(* PLC project Unnamed, Unknown Unnamed 1 *)
(* stored: creationDateTime 2021-11-19T07:51:07, modificationDateTime 2021-11-26T10:24:18 *)

PROGRAM program0
  VAR
    Start : BOOL;
    Stop : BOOL;
    ConveyorBelt : BOOL;
    A : BOOL;
    B : BOOL;
    TON0 : TON;
    TON1 : TON;
    DetectCan : BOOL;
    DetectCap : BOOL;
    Wait1 : BOOL;
    TON2 : TON;
    Stop1 : BOOL;
    Detect : BOOL;
    ShootInkJet : BOOL;
    Wait2 : BOOL;
    TON3 : TON;
    Stop2 : BOOL;
    CountCan : BOOL;
    CTU0 : CTU;
    StartPalletizer : BOOL;
    CTU1 : CTU;
  END_VAR
  VAR  (* added by the conversion: wires and edge detectors of the diagram *)
    R_TRIG1 : R_TRIG;
    R_TRIG2 : R_TRIG;
  END_VAR

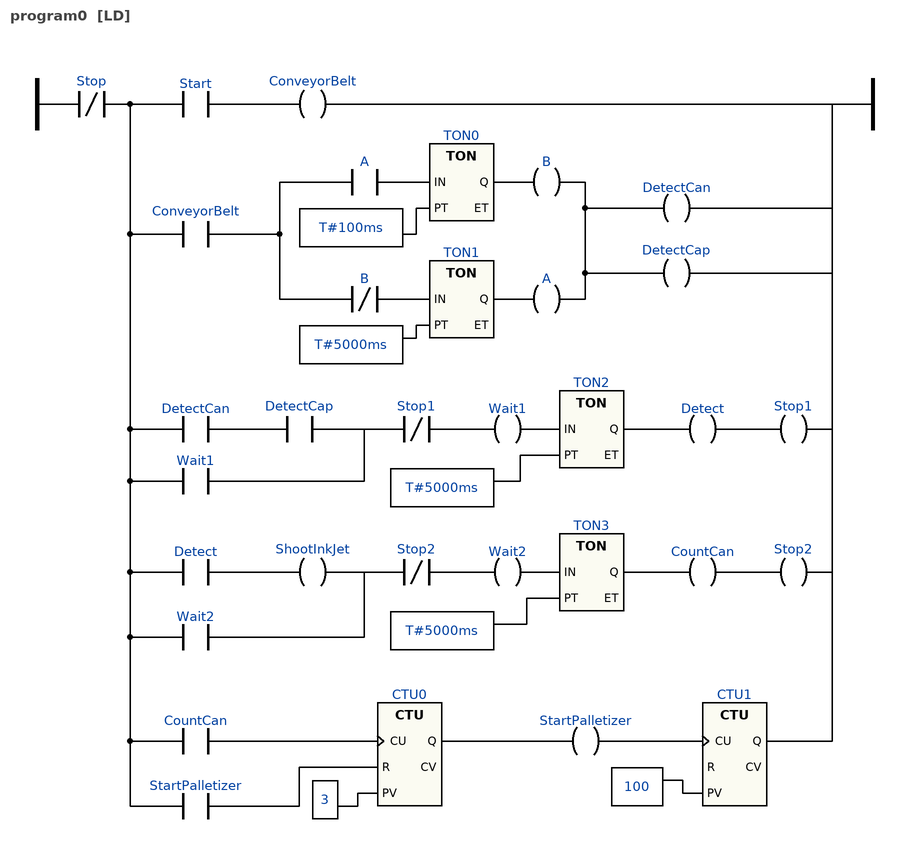
(* LD diagram, written out as Structured Text *)
ConveyorBelt := NOT Stop AND Start;
TON0(IN := NOT Stop AND ConveyorBelt AND A, PT := T#100ms);
B := TON0.Q;
TON1(IN := NOT Stop AND ConveyorBelt AND NOT B, PT := T#5000ms);
DetectCan := TON0.Q OR TON1.Q;
DetectCap := TON0.Q OR TON1.Q;
A := TON1.Q;
Wait1 := NOT Stop AND (DetectCan AND DetectCap OR Wait1) AND NOT Stop1;
TON2(IN := NOT Stop AND (DetectCan AND DetectCap OR Wait1) AND NOT Stop1, PT := T#5000ms);
Detect := TON2.Q;
Stop1 := TON2.Q;
ShootInkJet := NOT Stop AND Detect;
Wait2 := NOT Stop AND (Detect OR Wait2) AND NOT Stop2;
TON3(IN := NOT Stop AND (Detect OR Wait2) AND NOT Stop2, PT := T#5000ms);
CountCan := TON3.Q;
Stop2 := TON3.Q;
R_TRIG1(CLK := NOT Stop AND CountCan);
CTU0(CU := R_TRIG1.Q, R := NOT Stop AND StartPalletizer, PV := 3);
StartPalletizer := CTU0.Q;
R_TRIG2(CLK := CTU0.Q);
CTU1(CU := R_TRIG2.Q, PV := 100);
END_PROGRAM

CONFIGURATION Config0
  RESOURCE Res0 ON PLC
    TASK task0(INTERVAL := T#20ms, PRIORITY := 0);
    PROGRAM instance0 WITH task0 : program0;
  END_RESOURCE
END_CONFIGURATION
